// TIA Portal V19 export
TYPE "LEXCHANGETRAY_typePlasticWorkStationIoSignalProcessValues"
// simulated: Bool
// inspectionAfterPlasticTrayJackingU2EM5: Bool
// plasticTrayTrayInplaceDetectionU2EM5: Bool
// plasticTrayLiftingCylinderworkingPositionDetectionU2EM5_1: Bool
// plasticTrayFeedingDetectionU2EM5: Bool
// inspectionBeforePlasticTrayJackingU2EM5: Bool
// plasticTrayLiftingCylinderHomePositionDetectionU2EM5_1: Bool
// scapegoat1SignalU2EM5: Bool
// scapegoat2SignalU2EM5: Bool
// stored: Access Published
   STRUCT
      simulated : Bool;
      inspectionAfterPlasticTrayJackingU2EM5 : Bool;
      plasticTrayTrayInplaceDetectionU2EM5 : Bool;
      plasticTrayLiftingCylinderworkingPositionDetectionU2EM5_1 : Bool;
      plasticTrayFeedingDetectionU2EM5 : Bool;
      inspectionBeforePlasticTrayJackingU2EM5 : Bool;
      plasticTrayLiftingCylinderHomePositionDetectionU2EM5_1 : Bool;
      scapegoat1SignalU2EM5 : Bool;
      scapegoat2SignalU2EM5 : Bool;
   END_STRUCT;
END_TYPE
